(* CODESYS project MQTT_Client.library
   Author: Stefan Roßmann
   Title: MQTT Client Library
   Version: 3.5.13.27
   Placeholder: MQTT Client
   DocFormat: reStructuredText
   Description: MQTT Client library
   Company: Stefan Roßmann Engineering Solutions
   LanguageModelAttribute: qualified-access-only
   DefaultNamespace: MQTT_Client

Project tree, tasks and I/O mapping:
  libraries: SysSocket23, * (System); Standard, * (System); CAA Memory, * (CAA Technical Workgroup)
  Projektinformationen/
    function GetVersion [ST]
    function GetCompany [ST]
    function GetTitle [ST]
    function GetTextProperty2 [ST]
    function GetTextProperty [ST]
    function GetBooleanProperty [ST]
    function GetVersionProperty [ST]
    function GetNumberProperty [ST]
  00000000-0000-0000-0000-000000000000|Z:\Pictures\Rossmann-Engineering_Logo.png
  MQTT_Client/
    Structs/
    Types/
    Function Blocks/
      function block FB_CalculateRemainingLength [ST]
      function block FB_DecodeRemainingLength [ST]
      function block FB_MQTTClient [ST]
      function block FB_Random [ST]
      function block FB_TimingFlag [ST]
    Functions/
      function FC_AddKeyValueToJSON [ST]
      function FC_CreateJSON [ST]
    Images/
      Rossmann-Engineering_Logo
    Interfaces/
    GlobalConstants/
    Enums/
    GlobalVariables/
      global variables GVL_thingsboard
  Bibliotheksinformation/
    function IsLibReleased [ST]
    function GetLibVersion [ST]
    function GetLibVersionNumber [ST]
*)

// MQTT_Client/GlobalVariables/GVL_thingsboard
{attribute 'qualified_only'}
VAR_GLOBAL
	ars_key: ARRAY [0..1000] OF STRING(255);
	ars_value: ARRAY [0..1000] OF STRING(255);
	iCount: INT;
END_VAR

// Projektinformationen/GetVersion
// This function has been automatically generated from the project information.
{attribute 'signature_flag' := '1073741824'}
{attribute 'register_in_runtime'}
FUNCTION GetVersion : VERSION
VAR_INPUT
	
END_VAR

GetVersion.uiMajor := 3;
GetVersion.uiMinor := 5;
GetVersion.uiServicePack := 13;
GetVersion.uiPatch := 27;

END_FUNCTION

// MQTT_Client/Function Blocks/FB_CalculateRemainingLength
{attribute 'hide'}
FUNCTION_BLOCK FB_CalculateRemainingLength
VAR_INPUT
	wNumberOfBytes: WORD;
	
END_VAR
VAR_OUTPUT
	iNumberOfBytesRemianingLengthField: INT;
	arbyRemainingBytesField: ARRAY[0..3] OF BYTE;
END_VAR
VAR
	bEncodedByte: BYTE;
	wValue: WORD;
	iCount: INT;
END_VAR

wValue:=wNumberOfBytes;
iCount := 0;
REPEAT
	bEncodedByte:=UINT_TO_BYTE(wValue MOD 128);
	wValue:=wVALUE / 128;
	
	IF (wVALUE > 0) THEN
		bEncodedByte := (bEncodedByte OR 128);
	END_IF
	arbyRemainingBytesField[iCount] := bEncodedByte;
	iCount := iCount + 1;

UNTIL (wValue <= 0)
END_REPEAT;
iNumberOfBytesRemianingLengthField:=iCount;

END_FUNCTION_BLOCK

// Projektinformationen/GetCompany
// This function has been automatically generated from the project information.
{attribute 'signature_flag' := '1073741824'}
{attribute 'register_in_runtime'}
FUNCTION GetCompany : WSTRING
VAR_INPUT
	
END_VAR

GetCompany := "Stefan Roßmann Engineering Solutions";

END_FUNCTION

// Bibliotheksinformation/IsLibReleased
// This function has been automatically generated from the project information.
FUNCTION IsLibReleased : BOOL
VAR_INPUT
	
END_VAR

IsLibReleased := FALSE;

END_FUNCTION

// Projektinformationen/GetTitle
// This function has been automatically generated from the project information.
{attribute 'signature_flag' := '1073741824'}
{attribute 'register_in_runtime'}
FUNCTION GetTitle : WSTRING
VAR_INPUT
	
END_VAR

GetTitle := "MQTT Client Library";

END_FUNCTION

// MQTT_Client/Function Blocks/FB_DecodeRemainingLength
FUNCTION_BLOCK FB_DecodeRemainingLength
VAR_INPUT
	abyRemainingLengthField: ARRAY[0..3] OF BYTE;
END_VAR
VAR_OUTPUT
	uiRemeiningLength: UINT;
END_VAR
VAR
	multiplier: UINT;
	value: UINT;
	iCount: INT;
END_VAR

multiplier := 1;
value := 0;
iCount :=0;
REPEAT
	value := value + (abyRemainingLengthField [iCount] AND 127)*multiplier;
	multiplier := multiplier * 128;
UNTIL ((abyRemainingLengthField [iCount] AND 128) <> 0)
END_REPEAT;
uiRemeiningLength:=value;

END_FUNCTION_BLOCK

// MQTT_Client/Function Blocks/FB_MQTTClient
//{attribute 'hide_all_locals'}
//This Function Block implements an MQTT Client
//Allows to Publish Messages to an MQTT-Broker
//Supported:
//Retain Messages
//Optional Last Will and Testament
//Optional Username and Password authentication
//QoS0: (At most once)
FUNCTION_BLOCK FB_MQTTClient
VAR_INPUT
	// Enables the Function block, The rising Edge of this Input automatically connects to the MQTT Broker - Standard: TRUE
	i_xEnable: BOOL := TRUE;
	// IP-Address (example: 192.168.178.101) or Webaddress (www.mqtt-dashboard.com) of the MQTT-Broker
	i_sBrokerAddress: STRING := 'www.mqtt-dashboard.com';
	// Port of the MQTT-Broker - Standard: 1883
	i_uiPort: UINT := 1883;
	// Optional Username if required
	i_sUsername: STRING := '';
	// Optional Password if required
	i_sPassword: STRING := '';
	// Last Will Topic if required (Automatically enables Will Message if changed) - otherwise leave untouched
	i_sWillTopic: STRING := '';
	// Last Will Message if required - otherwise leave untouched
	i_sWillMessage: STRING := '';
	// Retain Last Will Message, if required Standard: FALSE - otherwise leave untouched 
	i_sWillRetain: BOOL := FALSE;	
	// Automatically try to reconnect after an Exception - Standard: TRUE
	i_xAutoReconnect: BOOL := TRUE;
	// PayLoad to Publish
	i_sPayload: STRING (255) := 'Hello MQTT-Broker from CoDeSys';
	// Topic to Publish to
	i_sTopicPublish: STRING := 'CoDeSys';
	// Topic to Subscribe
	i_sTopicSubscribe: STRING := 'CoDeSys';
	// Retain Flag Forces the Broker to Retain the Last Mesage - Standard: TRUE
	i_xRetain: BOOL := TRUE;
	// Publish the Payload to the Topic of the MQTT-Broker
	i_xPublish: BOOL:=FALSE;
	// Subscribe to the Topic given to the Input i_sTopicSubscribe
	i_xSubscribe: BOOL:=FALSE;
	// ClientID. If this Input is set we send the ClientID from the FB Input, otherise Random
	i_sClientID: STRING:='12345678';
END_VAR
VAR_OUTPUT
	// Message Received from a subsribed Topic
	q_sLastReceivedMessage: STRING(1024);
	// Topic Message Received
	q_sLastReceivedMessageTopic: STRING;	
	// Last 25 Received Messages
	q_arsLastReceivedMessages: ARRAY [0..24] OF STRING(1024);
	// Last 25 Topics Received
	q_arsLastReceivedMessageTopics: ARRAY [0..24] OF STRING;	
	// Message Received Notification
	q_xReceivedMessageNotification: BOOL;
	// Diag Message
	q_sDiagMsg: STRING;
	// Current State of the Function Block
	q_udiState: UDINT;
	// Error Flag
	q_xError: BOOL;
END_VAR
VAR
	R_TRIG_Enable: R_TRIG;
	diSocket : DINT ; 
	diAddressFamily : DINT := SOCKET_AF_INET; 
	diType : DINT := SOCKET_STREAM;
	diProtocol : DINT := SOCKET_IPPROTO_TCP;

	
	sockAddr : SOCKADDRESS;
	
	xResult : BOOL;
	outBuffer: ARRAY[0..1000] OF BYTE;
	inBuffer: ARRAY[0..1000] OF BYTE;
	diResult: DINT;
	IFB_CalculateRemainingLength: FB_CalculateRemainingLength;
	IFB_Random: ARRAY[0..9] OF FB_Random;
	wKeepAlive: WORD := 60;
	IoCtlParameter : DINT := 1;

	R_TRIG_Publish: R_TRIG;
	R_TRIG_Subscribe: R_TRIG;

	uiYear:UINT;
	uiMonth: UINT;
	uiDay: UINT;
	uiHour: UINT;
	uiMinute: UINT;
	uiSecond: UINT;
	
	TON_TimeOut: ton;
	wTimeOutValue: WORD;
	udiLastState: UDINT;
	
	xResultDisconnect: BOOL;
	QI: INT;
	
	iIndexCount: INT;
	wPacketIdentifierCount: WORD :=0;
	uiPayLoadLength: uint;
	
	xPublish: BOOL;
	xSubscribe: BOOL;
	
	i: INT;
END_VAR

//Read Clock
//IFBGetDateTime(xExecute:=TRUE);
(*DTU.DTSplit(dtDateAndTime:=IFBGetDateTime.dtDateAndTime,
			puiYear:=ADR(uiYear),
			puiMonth:=ADR(uiMonth),
			puiDay:=ADR(uiDay),
			puiHour:=ADR(uiHour),
			puiMinute:=ADR(uiMinute),
			puiSecond:=ADR(uiSecond));*)
			

IFB_Random[0](A:=21345,B:=36215,V:=uiSecond);
IFB_Random[1](A:=42784,B:=926432,V:=uiSecond);
IFB_Random[2](A:=87654,B:=23456,V:=uiSecond);
IFB_Random[3](A:=76543,B:=12345,V:=uiSecond);
IFB_Random[4](A:=3456543234,B:=54321234,V:=uiSecond);
IFB_Random[5](A:=763435,B:=121234,V:=uiSecond);
IFB_Random[6](A:=897,B:=434321,V:=uiSecond);
IFB_Random[7](A:=345654332,B:=77765,V:=uiSecond);
IFB_Random[8](A:=21234,B:=8654,V:=uiSecond);
IFB_Random[9](A:=2354,B:=3123,V:=uiSecond);

R_TRIG_Enable(CLK:=i_xEnable);
R_TRIG_Publish(CLK:=i_xPublish);
R_TRIG_Subscribe(CLK:=i_xSubscribe);

IF (R_TRIG_Publish.Q) THEN
	xPublish:=TRUE;
END_IF

IF (R_TRIG_Subscribe.Q) THEN
	xSubscribe:=TRUE;
END_IF



CASE q_udiState OF
	
//0: Wait for Enable
0: 	wTimeOutValue:=0;
	IF (R_TRIG_Enable.Q) THEN
		sockAddr.sin_addr := 0;
	END_IF
		

	IF (NOT q_xError) THEN	
		q_sDiagMsg:='Wait for Enable';
	END_IF
	IF (R_TRIG_Enable.Q OR (i_xAutoReconnect AND q_xError)) THEN
		q_xError := FALSE;
		q_udiState:=5;
	END_IF

//5: Create Socket
5:  diSocket := SysSockCreate(diAddressFamily, diType, diProtocol);
	SysSockIoctl(diSocket, SOCKET_FIONBIO, ADR(IoCtlParameter));	//Send socket to non blocking
	q_sDiagMsg:='Create Socket';
	wTimeOutValue:=500;
	IF (diSocket > 0) THEN
		q_udiState := 10;
	END_IF
	IF (TON_TimeOut.Q) THEN
		q_udiState:=0;	
		q_xError := TRUE;
		q_sDiagMsg:='Creating Socket Timed Out';
	END_IF
	

10: 
//10: Connect to TCP Server
	IF (sockAddr.sin_addr = 0) THEN
		sockAddr.sin_family := SOCKET_AF_INET; 
		IF (right(i_sBrokerAddress,1) = '0' OR right(i_sBrokerAddress,1) = '1' OR right(i_sBrokerAddress,1) = '2' OR right(i_sBrokerAddress,1) = '3' OR right(i_sBrokerAddress,1) = '4'
			OR right(i_sBrokerAddress,1) = '5' OR right(i_sBrokerAddress,1) = '6' OR right(i_sBrokerAddress,1) = '7' OR right(i_sBrokerAddress,1) = '8' OR right(i_sBrokerAddress,1) = '9') THEN
			sockAddr.sin_addr := SysSockInetAddr(i_sBrokerAddress); 
		ELSE
			sockAddr.sin_addr := SysSockGetHostByName(i_sBrokerAddress);
			
			
		END_IF
	END_IF
	 
	sockAddr.sin_port :=  SysSockHtons(i_uiPort);
	wTimeOutValue:=1000;
	xResult := SysSockConnect(diSocket, ADR(sockAddr), SIZEOF(sockAddr));
	q_sDiagMsg:='Connect to TCP-Server';
	IF (xResult) THEN
		q_udiState:=15;	
	END_IF
	IF (TON_TimeOut.Q) THEN
		q_udiState:=90;	
		q_xError := TRUE;
		q_sDiagMsg:='Connecting to TCP-Server Timed out';
	END_IF

//15: Initialize OutBuffer
15: outBuffer[0] := 16;		//MQTT Control Packet Type
	wTimeOutValue:=0;
	//Calculate the length - Length must be 10 + Payload (We use 10 bytes client ID)
	IFB_CalculateRemainingLength(wNumberOfBytes:=10 + 2 + len(i_sClientID) + (2+len(i_sUsername)) * BOOL_TO_INT(i_sUsername <> '') + (2+len(i_sPassword)) * BOOL_TO_INT(i_sPassword <> '')  + (2+len(i_sWillTopic)) * BOOL_TO_INT(i_sWillTopic <> '') + (2+len(i_sWillMessage)) * BOOL_TO_INT(i_sWillMessage <> '') );

	outBuffer[1] := IFB_CalculateRemainingLength.arbyRemainingBytesField[0];		
	outBuffer[2] := IFB_CalculateRemainingLength.arbyRemainingBytesField[1];
	outBuffer[3] := IFB_CalculateRemainingLength.arbyRemainingBytesField[2];
	outBuffer[4] := IFB_CalculateRemainingLength.arbyRemainingBytesField[3];

	outBuffer[1 + IFB_CalculateRemainingLength.iNumberOfBytesRemianingLengthField] := 0;		//Length MSB (0)
	outBuffer[2	+ IFB_CalculateRemainingLength.iNumberOfBytesRemianingLengthField] := 4;		//Length LSB (1)
	outBuffer[3	+ IFB_CalculateRemainingLength.iNumberOfBytesRemianingLengthField] := 77;		//'M'
	outBuffer[4	+ IFB_CalculateRemainingLength.iNumberOfBytesRemianingLengthField] := 81;		//'Q'
	outBuffer[5	+ IFB_CalculateRemainingLength.iNumberOfBytesRemianingLengthField] := 84;		//'T'
	outBuffer[6	+ IFB_CalculateRemainingLength.iNumberOfBytesRemianingLengthField] := 84;		//'T'
	outBuffer[7	+ IFB_CalculateRemainingLength.iNumberOfBytesRemianingLengthField] := 4;		//Protocol Level (4)

	outBuffer[8	+ IFB_CalculateRemainingLength.iNumberOfBytesRemianingLengthField] := 2 OR (BOOL_TO_BYTE(i_sPassword <> '') * 64) 
																						OR (BOOL_TO_BYTE(i_sUsername <> '') * 128) 
																						OR (BOOL_TO_BYTE(i_sWillTopic <> '') * 4)
																						OR (BOOL_TO_BYTE(i_sWillRetain) * 32);	
																							//Connect Flags: 0: Reserved; 1: Clean Session
																							//2: Will Flag; 3+4: Will QoS; 5: Will Retain; 6: Password Flas, 7: Username Flag

	wKeepAlive := 60;
	outBuffer[9	+ IFB_CalculateRemainingLength.iNumberOfBytesRemianingLengthField] := WORD_TO_BYTE(SHR(wKeepAlive,8));		//Keep Alive MSB
	outBuffer[10+ IFB_CalculateRemainingLength.iNumberOfBytesRemianingLengthField] := WORD_TO_BYTE(wKeepAlive);		//Keep Alive LSB
	iIndexCount:=11;
	IF (i_sClientID = '12345678') THEN
		//Auto Generated ClientID
		outBuffer[11+ IFB_CalculateRemainingLength.iNumberOfBytesRemianingLengthField] := 0;//REAL_TO_BYTE(IFB_Random[0].dwRandom);
		outBuffer[12+ IFB_CalculateRemainingLength.iNumberOfBytesRemianingLengthField] := 8;//REAL_TO_BYTE(IFB_Random[1].dwRandom);
		outBuffer[13+ IFB_CalculateRemainingLength.iNumberOfBytesRemianingLengthField] := REAL_TO_BYTE(IFB_Random[2].dwRandom);
		outBuffer[14+ IFB_CalculateRemainingLength.iNumberOfBytesRemianingLengthField] := REAL_TO_BYTE(IFB_Random[3].dwRandom);
		outBuffer[15+ IFB_CalculateRemainingLength.iNumberOfBytesRemianingLengthField] := REAL_TO_BYTE(IFB_Random[4].dwRandom);
		outBuffer[16+ IFB_CalculateRemainingLength.iNumberOfBytesRemianingLengthField] := REAL_TO_BYTE(IFB_Random[5].dwRandom);
		outBuffer[17+ IFB_CalculateRemainingLength.iNumberOfBytesRemianingLengthField] := REAL_TO_BYTE(IFB_Random[6].dwRandom);
		outBuffer[18+ IFB_CalculateRemainingLength.iNumberOfBytesRemianingLengthField] := REAL_TO_BYTE(IFB_Random[7].dwRandom);
		outBuffer[19+ IFB_CalculateRemainingLength.iNumberOfBytesRemianingLengthField] := REAL_TO_BYTE(IFB_Random[8].dwRandom);
		outBuffer[20+ IFB_CalculateRemainingLength.iNumberOfBytesRemianingLengthField] := REAL_TO_BYTE(IFB_Random[9].dwRandom);
		iIndexCount:=21;
	ELSE
		//ClientID from FB Input		
		outBuffer[11+ IFB_CalculateRemainingLength.iNumberOfBytesRemianingLengthField] := INT_TO_BYTE(SHR(len(i_sClientID),8));//REAL_TO_BYTE(IFB_Random[0].dwRandom);
		outBuffer[12+ IFB_CalculateRemainingLength.iNumberOfBytesRemianingLengthField] := INT_TO_BYTE(len(i_sClientID));//REAL_TO_BYTE(IFB_Random[1].dwRandom);
		iIndexCount := iIndexCount + 2;
		MEM.MemMove(ADR(i_sClientID),ADR(outBuffer[iIndexCount	+ IFB_CalculateRemainingLength.iNumberOfBytesRemianingLengthField]),len(i_sClientID));
		iIndexCount:=iIndexCount+len(i_sClientID);
	END_IF
	
	//iIndexCount:=21;
	//Set Will Topic
	IF (i_sWillTopic <> '') THEN
		outBuffer[iIndexCount+ IFB_CalculateRemainingLength.iNumberOfBytesRemianingLengthField] := INT_TO_BYTE(SHR(len(i_sWillTopic),8));		//Length MSB
		iIndexCount:=iIndexCount+1;
		outBuffer[iIndexCount+ IFB_CalculateRemainingLength.iNumberOfBytesRemianingLengthField] := INT_TO_BYTE(len(i_sWillTopic));				//Length MSB
		iIndexCount:=iIndexCount+1;
		MEM.MemMove(ADR(i_sWillTopic),ADR(outBuffer[iIndexCount	+ IFB_CalculateRemainingLength.iNumberOfBytesRemianingLengthField]),len(i_sWillTopic));
		iIndexCount:=iIndexCount+len(i_sWillTopic);
	END_IF
	
	//Set Will Message
	IF (i_sWillMessage <> '') THEN
		outBuffer[iIndexCount+ IFB_CalculateRemainingLength.iNumberOfBytesRemianingLengthField] := INT_TO_BYTE(SHR(len(i_sWillMessage),8));		//Length MSB
		iIndexCount:=iIndexCount+1;
		outBuffer[iIndexCount+ IFB_CalculateRemainingLength.iNumberOfBytesRemianingLengthField] := INT_TO_BYTE(len(i_sWillMessage));				//Length MSB
		iIndexCount:=iIndexCount+1;
		MEM.MemMove(ADR(i_sWillMessage),ADR(outBuffer[iIndexCount	+ IFB_CalculateRemainingLength.iNumberOfBytesRemianingLengthField]),len(i_sWillMessage));
		iIndexCount:=iIndexCount+len(i_sWillMessage);
	END_IF
	
	//Set Username
	IF (i_sUsername <> '') THEN
		outBuffer[iIndexCount+ IFB_CalculateRemainingLength.iNumberOfBytesRemianingLengthField] := INT_TO_BYTE(SHR(len(i_sUsername),8));		//Length MSB
		iIndexCount:=iIndexCount+1;
		outBuffer[iIndexCount+ IFB_CalculateRemainingLength.iNumberOfBytesRemianingLengthField] := INT_TO_BYTE(len(i_sUsername));				//Length MSB
		iIndexCount:=iIndexCount+1;
		MEM.MemMove(ADR(i_sUsername),ADR(outBuffer[iIndexCount	+ IFB_CalculateRemainingLength.iNumberOfBytesRemianingLengthField]),len(i_sUsername));
		iIndexCount:=iIndexCount+len(i_sUsername);
	END_IF
	
	//Set Password
	IF (i_sPassword <> '') THEN
		outBuffer[iIndexCount+ IFB_CalculateRemainingLength.iNumberOfBytesRemianingLengthField] := INT_TO_BYTE(SHR(len(i_sPassword),8));		//Length MSB
		iIndexCount:=iIndexCount+1;
		outBuffer[iIndexCount+ IFB_CalculateRemainingLength.iNumberOfBytesRemianingLengthField] := INT_TO_BYTE(len(i_sPassword));				//Length MSB
		iIndexCount:=iIndexCount+1;
		MEM.MemMove(ADR(i_sPassword),ADR(outBuffer[iIndexCount	+ IFB_CalculateRemainingLength.iNumberOfBytesRemianingLengthField]),len(i_sPassword));
		iIndexCount:=iIndexCount+len(i_sUsername);
	END_IF
	
	q_sDiagMsg:='Initialize Out-Buffer';
	q_udiState:=20;

//20: Send Connect	
20:		
	diResult := SysSockSend(diSocket, ADR(outBuffer), 11 + 2 + len(i_sClientID)+ IFB_CalculateRemainingLength.iNumberOfBytesRemianingLengthField+(2+len(i_sUsername)) * BOOL_TO_INT(i_sUsername <> '') + (2+len(i_sPassword)) * BOOL_TO_INT(i_sPassword <> '') + (2+len(i_sWillTopic)) * BOOL_TO_INT(i_sWillTopic <> '') + (2+len(i_sWillMessage)) * BOOL_TO_INT(i_sWillMessage <> ''), 0);
	q_sDiagMsg:='Connect to MQTT-Broker';
	wTimeOutValue:=1000;
	IF (diResult > 0) THEN 
		q_udiState:=30;	
	END_IF
	IF (TON_TimeOut.Q) THEN
		q_udiState:=0;	
		q_xError := TRUE;
		q_sDiagMsg:='Connecting to MQTT-Broker (MQTT Control Packet) Timed out';
	END_IF

//30: Wait for CONNACK from Broker
30: diResult := SysSockRecv(diSocket:=diSocket,pbyBuffer:=ADR(inBuffer),diBufferSize:=500,diFlags:=0);
	q_sDiagMsg:='Wait for Connack from Broker';
	wTimeOutValue:=1000;
	IF (diResult > 0) THEN
		q_udiState:=40;	
		diResult:=0;
	END_IF
	IF (TON_TimeOut.Q) THEN
		q_udiState:=90;	
		q_xError := TRUE;
		q_sDiagMsg:='Waiting for "Connack" from MQTT-Broker Timed out';
	END_IF

//40: Analyze CONNACK
40:	q_sDiagMsg:='Analyze connack';
	wTimeOutValue:=0;
	IF (inBuffer[0] = 32 AND inBuffer[3] = 0) THEN
		q_udiState := 60;
	ELSE
		//Return code repsone (2nd Byte): 
		//0: Connection Accepted
		//1: Connection Refused, unacceptable protocol version
		IF (inBuffer[3] = 1) THEN
			q_sDiagMsg:='Connection Refused, unacceptable protocol version';
		END_IF
		//2: Connection Refused, identifier rejected
		IF (inBuffer[3] = 2) THEN
			q_sDiagMsg:='Connection Refused, identifier rejected';
		END_IF
		//3: Connection Refused, Server unavailable
		IF (inBuffer[3] = 3) THEN
			q_sDiagMsg:='Connection Refused, Server unavailable';
		END_IF		
		//4: Connection Refused, bad Username or passworrd
		IF (inBuffer[3] = 4) THEN
			q_sDiagMsg:='Connection Refused, bad Username or password';
		END_IF	
		//5: Connection Refused, not autorized
		IF (inBuffer[3] = 5) THEN
			q_sDiagMsg:='Connection Refused, not autorized';
		END_IF	
		q_xError := TRUE;
		q_udiState := 90;	
	END_IF
	
//60: Wait for Publish or Disconnect (Enable low)
60:	q_sDiagMsg:='Wait for Publish or Subscribe or Disconnect (Enable low)';
	wTimeOutValue:=0;
	q_xReceivedMessageNotification:= FALSE;
	diResult := SysSockRecv(diSocket:=diSocket,pbyBuffer:=ADR(inBuffer),diBufferSize:=500,diFlags:=0);
	IF (xPublish) THEN
		xPublish:=FALSE;
		q_udiState := 70;	
	END_IF
	IF (xSubscribe) THEN
		xSubscribe:=FALSE;
		q_udiState := 65;	
	END_IF
	IF (NOT i_xEnable) THEN
		q_udiState := 80;	
	END_IF
	IF (diResult > 0) THEN
		
		q_xReceivedMessageNotification:= TRUE;
		q_udiState := 63;	
		
	END_IF
	
//Analyze Publish Message from Broker
63: q_sDiagMsg:='Analyze Publish Message from Broker';
	wTimeOutValue:=0;

	IFB_CalculateRemainingLength(wNumberOfBytes:=DINT_TO_WORD(diResult-2));
	uiPayLoadLength:=DINT_TO_UINT(diResult) - SHL(BYTE_TO_UINT(inBuffer[IFB_CalculateRemainingLength.iNumberOfBytesRemianingLengthField+1]),8) - (inBuffer[IFB_CalculateRemainingLength.iNumberOfBytesRemianingLengthField+2]) - 4;
	mem.MemFill(ADR(q_sLastReceivedMessage),80,0);
	mem.MemFill(ADR(q_sLastReceivedMessageTopic),80,0);
	MEM.MemMove(ADR(inBuffer[diResult-uiPayLoadLength+1]),ADR(q_sLastReceivedMessage),uiPayLoadLength);
	MEM.MemMove(ADR(inBuffer[IFB_CalculateRemainingLength.iNumberOfBytesRemianingLengthField+3]),ADR(q_sLastReceivedMessageTopic),DINT_TO_UINT(diResult)-uiPayLoadLength-IFB_CalculateRemainingLength.iNumberOfBytesRemianingLengthField-3);
	
	FOR i := 24 TO 1 BY -1 DO		
		q_arsLastReceivedMessageTopics[i] := q_arsLastReceivedMessageTopics[i-1];	
		q_arsLastReceivedMessages[i] := q_arsLastReceivedMessages[i-1];	
	END_FOR
	
	q_arsLastReceivedMessageTopics[0]:=q_sLastReceivedMessageTopic;
	q_arsLastReceivedMessages[0]:=q_sLastReceivedMessage;
	
	diResult:=0;
	q_udiState := 60;	
	
//65: Subscribe to Topic
65: q_sDiagMsg:='Subscribe to Topic';
	wTimeOutValue:=1000;
	//Calculate the length - Length of Variable Header + Length of Payload
	IFB_CalculateRemainingLength(wNumberOfBytes:=len(i_sTopicSubscribe) +5);
	outBuffer[0] := 130;		//MQTT Control Packet Type
	
	outBuffer[1] := IFB_CalculateRemainingLength.arbyRemainingBytesField[0];		
	outBuffer[2] := IFB_CalculateRemainingLength.arbyRemainingBytesField[1];
	outBuffer[3] := IFB_CalculateRemainingLength.arbyRemainingBytesField[2];
	outBuffer[4] := IFB_CalculateRemainingLength.arbyRemainingBytesField[3];
	
	wPacketIdentifierCount:=wPacketIdentifierCount + 1;
	IF (wPacketIdentifierCount = 0) THEN
		wPacketIdentifierCount:=1;
	END_IF
	
	outBuffer[1 + IFB_CalculateRemainingLength.iNumberOfBytesRemianingLengthField] := INT_TO_BYTE(SHR(wPacketIdentifierCount,8));		//Packet Identifier MSB
	outBuffer[2	+ IFB_CalculateRemainingLength.iNumberOfBytesRemianingLengthField] := INT_TO_BYTE(wPacketIdentifierCount);				//Packet Identifier LSB
	
	outBuffer[3 + IFB_CalculateRemainingLength.iNumberOfBytesRemianingLengthField] := INT_TO_BYTE(SHR(len(i_sTopicSubscribe),8));		//Length MSB
	outBuffer[4	+ IFB_CalculateRemainingLength.iNumberOfBytesRemianingLengthField] := INT_TO_BYTE(len(i_sTopicSubscribe));		//Length LSB
	MEM.MemMove(ADR(i_sTopicSubscribe),ADR(outBuffer[5	+ IFB_CalculateRemainingLength.iNumberOfBytesRemianingLengthField]),len(i_sTopicSubscribe));
	
	outBuffer[5	+ len(i_sTopicSubscribe) + IFB_CalculateRemainingLength.iNumberOfBytesRemianingLengthField] := 0;	
	diResult := SysSockSend(diSocket, ADR(outBuffer), (6 + len(i_sTopicSubscribe) + IFB_CalculateRemainingLength.iNumberOfBytesRemianingLengthField) , 0);
	IF (diResult > 0) THEN 
		
		q_udiState:=66;	
	END_IF	
	IF (TON_TimeOut.Q) THEN
		q_udiState:=90;	
		q_xError := TRUE;
		q_sDiagMsg:='Subscribe (MQTT Control Packet) Timed out';
	END_IF	
	
//66: Wait for SUBACK from Broker
66: diResult := SysSockRecv(diSocket:=diSocket,pbyBuffer:=ADR(inBuffer),diBufferSize:=500,diFlags:=0);
	q_sDiagMsg:='Wait for SUBACK from Broker';
	wTimeOutValue:=1000;
	IF (diResult > 0) THEN
		q_udiState:=67;	
		diResult:=0;
	END_IF
	IF (TON_TimeOut.Q) THEN
		q_udiState:=90;	
		q_xError := TRUE;
		q_sDiagMsg:='Waiting for "Suback" from MQTT-Broker Timed out';
	END_IF

//67: Analyze SUBACK
67:	q_sDiagMsg:='Analyze SUBACK';
	wTimeOutValue:=0;
	IF (inBuffer[diResult-1] < 16#80) THEN
		q_udiState := 60;
		diResult:=0;
	ELSE	
		q_udiState:=90;	
		q_xError := TRUE;
		q_sDiagMsg:='Suback Message reported Failure (Return code 0x80)';
	END_IF
		
	
	
//70: Publish Message
70: outBuffer[0] := 48 + BOOL_TO_BYTE(i_xRetain);		//MQTT Control Packet Type

	//Calculate the length - Length of Variable Header + Length of Payload
	IFB_CalculateRemainingLength(wNumberOfBytes:=len(i_sTopicPublish) + len(i_sPayload)+2);

	outBuffer[1] := IFB_CalculateRemainingLength.arbyRemainingBytesField[0];		
	outBuffer[2] := IFB_CalculateRemainingLength.arbyRemainingBytesField[1];
	outBuffer[3] := IFB_CalculateRemainingLength.arbyRemainingBytesField[2];
	outBuffer[4] := IFB_CalculateRemainingLength.arbyRemainingBytesField[3];

	outBuffer[1 + IFB_CalculateRemainingLength.iNumberOfBytesRemianingLengthField] := INT_TO_BYTE(SHR(len(i_sTopicPublish),8));		//Length MSB
	outBuffer[2	+ IFB_CalculateRemainingLength.iNumberOfBytesRemianingLengthField] := INT_TO_BYTE(len(i_sTopicPublish));		//Length LSB
	
	MEM.MemMove(ADR(i_sTopicPublish),ADR(outBuffer[3	+ IFB_CalculateRemainingLength.iNumberOfBytesRemianingLengthField]),len(i_sTopicPublish));

	MEM.MemMove(ADR(i_sPayload),ADR(outBuffer[3 + len(i_sTopicPublish)	+ IFB_CalculateRemainingLength.iNumberOfBytesRemianingLengthField]),len(i_sPayload));
	

	diResult := SysSockSend(diSocket, ADR(outBuffer), (len(i_sTopicPublish) + len(i_sPayload)+3+ IFB_CalculateRemainingLength.iNumberOfBytesRemianingLengthField) , 0);
	q_sDiagMsg:='Publish Message';
	wTimeOutValue:=1000;
	IF (diResult > 0) THEN 
		diResult:=0;
		q_udiState:=60;	
	END_IF	
	IF (TON_TimeOut.Q) THEN
		q_udiState:=90;	
		q_xError := TRUE;
		q_sDiagMsg:='Publishing Message (MQTT Control Packet) Timed out';
	END_IF

//80: Send "Disconnect"
80: outBuffer[0] := 224;		//MQTT Control Packet Type
	outBuffer[1] := 0;			//Remaining Length (0)
	diResult := SysSockSend(diSocket, ADR(outBuffer), 2 , 0);
	q_sDiagMsg:='Send Disconnect notification to server';
	wTimeOutValue:=1000;
	IF (diResult > 0) THEN 
		diResult:=0;
		q_udiState:=90;	
	END_IF	
	IF (TON_TimeOut.Q) THEN
		q_udiState:=90;	
		q_xError := TRUE;
		q_sDiagMsg:='Sending Disconnect to MQTT-Broker Timed out';
	END_IF	

//90: Disconnect Socket
90:	xResultDisconnect := SysSockClose(diSocket);
	IF (NOT q_xError) THEN
		q_sDiagMsg:='Close TCP Socket';
	END_IF
	wTimeOutValue:=1000;
	IF (xResultDisconnect) THEN 
		q_udiState:=0;	
	END_IF	
	IF (TON_TimeOut.Q) THEN
		q_udiState:=0;	
		q_xError := TRUE;
		q_sDiagMsg:='Closing TCP-Socket  Timed out';
	END_IF	
END_CASE

TON_TimeOut(IN:=(udiLastState=q_udiState) AND (wTimeOutValue <> 0) ,PT:=WORD_TO_TIME(wTimeOutValue));
udiLastState:=q_udiState;

END_FUNCTION_BLOCK

// MQTT_Client/Function Blocks/FB_Random
	{attribute 'hide'}
FUNCTION_BLOCK FB_Random
VAR_INPUT
	A: DWORD;
	B: DWORD;
	V: DWORD;
END_VAR
VAR_OUTPUT
	dwRandom: dword;
END_VAR
VAR
	dwValue1: DWORD;
	dwValue2: DWORD;
	M: DWORD;
	Q: DWORD;

END_VAR


Q:=Q+2;

M:=25;
dwRandom:=(A+V+B+Q) MOD M + 65;

END_FUNCTION_BLOCK

// Projektinformationen/GetTextProperty2
// This function has been automatically generated from the project information.
{attribute 'signature_flag' := '1073741824'}
{attribute 'register_in_runtime'}
FUNCTION GetTextProperty2 : POINTER TO WSTRING
VAR_INPUT
	stKey: WSTRING;
END_VAR

IF stKey = "Author" THEN
	GetTextProperty2 := ADR("Stefan Roßmann");
ELSIF stKey = "Company" THEN
	GetTextProperty2 := ADR("Stefan Roßmann Engineering Solutions");
ELSIF stKey = "DefaultNamespace" THEN
	GetTextProperty2 := ADR("MQTT_Client");
ELSIF stKey = "Description" THEN
	GetTextProperty2 := ADR("MQTT Client library");
ELSIF stKey = "DocFormat" THEN
	GetTextProperty2 := ADR("reStructuredText");
ELSIF stKey = "LanguageModelAttribute" THEN
	GetTextProperty2 := ADR("qualified-access-only");
ELSIF stKey = "Placeholder" THEN
	GetTextProperty2 := ADR("MQTT Client");
ELSIF stKey = "Project" THEN
	GetTextProperty2 := ADR("MQTT_Client");
ELSIF stKey = "Title" THEN
	GetTextProperty2 := ADR("MQTT Client Library");
ELSE
	GetTextProperty2 := ADR("");
END_IF

END_FUNCTION

// Projektinformationen/GetTextProperty
// This function has been automatically generated from the project information.
{attribute 'signature_flag' := '1073741824'}
{attribute 'register_in_runtime'}
FUNCTION GetTextProperty : WSTRING
VAR_INPUT
	stKey: WSTRING;
END_VAR

IF stKey = "Author" THEN
	GetTextProperty := "Stefan Roßmann";
ELSIF stKey = "Company" THEN
	GetTextProperty := "Stefan Roßmann Engineering Solutions";
ELSIF stKey = "DefaultNamespace" THEN
	GetTextProperty := "MQTT_Client";
ELSIF stKey = "Description" THEN
	GetTextProperty := "MQTT Client library";
ELSIF stKey = "DocFormat" THEN
	GetTextProperty := "reStructuredText";
ELSIF stKey = "LanguageModelAttribute" THEN
	GetTextProperty := "qualified-access-only";
ELSIF stKey = "Placeholder" THEN
	GetTextProperty := "MQTT Client";
ELSIF stKey = "Project" THEN
	GetTextProperty := "MQTT_Client";
ELSIF stKey = "Title" THEN
	GetTextProperty := "MQTT Client Library";
ELSE
	GetTextProperty := "";
END_IF

END_FUNCTION

// Projektinformationen/GetBooleanProperty
// This function has been automatically generated from the project information.
{attribute 'signature_flag' := '1073741824'}
{attribute 'register_in_runtime'}
FUNCTION GetBooleanProperty : BOOL
VAR_INPUT
	stKey: WSTRING;
END_VAR

IF stKey = "IsEndUserLibrary" THEN
	GetBooleanProperty := FALSE;
ELSIF stKey = "Released" THEN
	GetBooleanProperty := FALSE;
ELSE
	GetBooleanProperty := FALSE;
END_IF

END_FUNCTION

// Projektinformationen/GetVersionProperty
// This function has been automatically generated from the project information.
{attribute 'signature_flag' := '1073741824'}
{attribute 'register_in_runtime'}
FUNCTION GetVersionProperty : VERSION
VAR_INPUT
	stKey: WSTRING;
END_VAR

IF stKey = "Version" THEN
	GetVersionProperty.uiMajor := 3;
	GetVersionProperty.uiMinor := 5;
	GetVersionProperty.uiServicePack := 13;
	GetVersionProperty.uiPatch := 27;
ELSE
	GetVersionProperty.uiMajor := 0;
	GetVersionProperty.uiMinor := 0;
	GetVersionProperty.uiServicePack := 0;
	GetVersionProperty.uiPatch := 0;
END_IF

END_FUNCTION

// Bibliotheksinformation/GetLibVersion
// This function has been automatically generated from the project information.
FUNCTION GetLibVersion : VERSION
VAR_INPUT
	
END_VAR

GetLibVersion.uiMajor := 3;
GetLibVersion.uiMinor := 5;
GetLibVersion.uiServicePack := 13;
GetLibVersion.uiPatch := 27;

END_FUNCTION

// Projektinformationen/GetNumberProperty
// This function has been automatically generated from the project information.
{attribute 'signature_flag' := '1073741824'}
{attribute 'register_in_runtime'}
FUNCTION GetNumberProperty : DINT
VAR_INPUT
	stKey: WSTRING;
END_VAR

GetNumberProperty := 0;

END_FUNCTION

// Bibliotheksinformation/GetLibVersionNumber
// This function has been automatically generated from the project information.
FUNCTION GetLibVersionNumber : DWORD
VAR_INPUT
	
END_VAR

GetLibVersionNumber := 50662683;

END_FUNCTION

// MQTT_Client/Functions/FC_AddKeyValueToJSON
FUNCTION FC_AddKeyValueToJSON : bool
VAR_INPUT
	i_sKeyToAdd: STRING(255) := 'key';
	i_sValueToAdd: STRING(255) := '4711';
END_VAR
VAR
END_VAR

IF (GVL_thingsboard.iCount < 1000) THEN
	GVL_thingsboard.ars_key[GVL_thingsboard.iCount] := i_sKeyToAdd;
	GVL_thingsboard.ars_value[GVL_thingsboard.iCount] := i_sValueToAdd;
	GVL_thingsboard.iCount := GVL_thingsboard.iCount + 1;
END_IF

END_FUNCTION

// MQTT_Client/Functions/FC_CreateJSON
FUNCTION FC_CreateJSON : STRING (255)
VAR_INPUT
	i_xInitArrayAfterCreate: BOOL:=TRUE;
END_VAR
VAR
	i: INT;
	returnvalue : STRING (255);
END_VAR

returnvalue := '{';
FOR i := 0 TO (GVL_thingsboard.iCount - 1) BY 1 DO
	returnvalue := CONCAT (returnvalue,GVL_thingsboard.ars_key[i]);
	returnvalue := CONCAT (returnvalue,':');
	returnvalue := CONCAT (returnvalue,GVL_thingsboard.ars_value[i]);
	IF i <> (GVL_thingsboard.iCount - 1) THEN
		returnvalue := CONCAT (returnvalue,',');
	END_IF
	
END_FOR
returnvalue := CONCAT (returnvalue,'}');


IF i_xInitArrayAfterCreate THEN
	GVL_thingsboard.iCount := 0;
END_IF

FC_CreateJSON := returnvalue;

END_FUNCTION

// MQTT_Client/Function Blocks/FB_TimingFlag
FUNCTION_BLOCK FB_TimingFlag
VAR_INPUT
	i_tTimebase: TIME;
END_VAR
VAR_OUTPUT
	q_xTimingFlag: BOOL;
END_VAR
VAR
	TON_Timer1: TP;
	TON_Timer2: tP;
END_VAR

TON_Timer1(IN:=NOT TON_Timer2.Q, PT:=(i_tTimebase/2));
TON_Timer2(IN:=NOT TON_Timer1.Q, PT:=(i_tTimebase/2));
q_xTimingFlag:=TON_Timer1.Q;

END_FUNCTION_BLOCK
